// Mitsubishi GX Works2 project: project2 (1)   PLC: FX3G

// global labels: Global1
VAR_GLOBAL
  startday AT X007 : BOOL;
  lemonInput AT D1100 : REAL;
  raspberryInput AT D1110 : REAL;
  gummyBearInput AT D1130 : REAL;
  workLed AT Y007 : BOOL;
  fictivyStartday AT M5 : BOOL;
  emrgency AT X005 : BOOL;
  finishIngridiance AT M1 : BOOL;
  endDay AT M6 : BOOL;
  enoughIngredients AT M7 : BOOL;
  startDgima AT X001 : BOOL;
  analogInput1 AT D8280 : INT;
END_VAR
VAR_GLOBAL CONSTANT
  normalizationFactor : REAL := 400;
END_VAR
VAR_GLOBAL
  gumigumType AT D1502 : REAL;
  minRegularGumigum AT E0.0 : REAL;
  maxRegularGumigum AT E5.0 : REAL;
  regularGumigum AT M12 : BOOL;
  minPinukGumigum AT E6.0 : REAL;
  pinukGumigum AT M13 : BOOL;
  stabilizerInput AT D1120 : REAL;
END_VAR
VAR_GLOBAL CONSTANT
  minLemonRaspberryRegular : REAL := 35;
  minRaspberryRaspberryRegular : REAL := 280;
  minStabilizerRaspberryRegular : REAL := 35;
END_VAR
VAR_GLOBAL
  checkRaspberryRegular AT M2 : BOOL;
  checkLemonRegular AT M3 : BOOL;
END_VAR
VAR_GLOBAL CONSTANT
  minLemonLemonRegular : REAL := 420;
  minRaspberryLemonRegular : REAL;
  minStabilizerLemonRegular : REAL := 70;
  minLemonRaspberryPinuk : REAL := 105;
  minRaspberryRaspberryPinuk : REAL := 385;
  minStabilizerRaspberryPinuk : REAL := 70;
END_VAR
VAR_GLOBAL
  chechRaspberryPinuk AT M4 : BOOL;
END_VAR
VAR_GLOBAL CONSTANT
  minLemonLemonPinuk : REAL := 560;
  minRaspberryLemonPinuk : REAL;
  minStabilizerLemonPinuk : REAL := 140;
END_VAR
VAR_GLOBAL
  checkLemonPinuk AT M15 : BOOL;
  timer5Sec AT TC1 : BOOL;
END_VAR
VAR_GLOBAL CONSTANT
  fiveSec : INT := 50;
END_VAR
VAR_GLOBAL
  finishTimer AT TS1 : BOOL;
  iceCreamMaking AT Y000 : BOOL;
  coolContainer AT X002 : BOOL;
  timer8Sec AT TC3 : BOOL;
END_VAR
VAR_GLOBAL CONSTANT
  eightSec : INT := 80;
END_VAR
VAR_GLOBAL
  temp10Degrees AT X003 : BOOL;
  coolLed AT Y002 : BOOL;
END_VAR
VAR_GLOBAL CONSTANT
  gummyBearPinuk : REAL := 70;
  gummyBearRegular : REAL := 28;
END_VAR
VAR_GLOBAL
  onOffLed AT M16 : BOOL;
  timerRegularGummigum AT TC33 : BOOL;
END_VAR
VAR_GLOBAL CONSTANT
  OnOffRegular : INT := 30;
END_VAR
VAR_GLOBAL
  timerPinukGummigum AT TC55 : BOOL;
END_VAR
VAR_GLOBAL CONSTANT
  OnOffPinuk : INT := 50;
END_VAR
VAR_GLOBAL
  timerReset AT M17 : BOOL;
  timer1 AT TC10 : BOOL;
END_VAR
VAR_GLOBAL CONSTANT
  timeInterval : INT := 7;
END_VAR
VAR_GLOBAL
  endTimer1 AT TS10 : BOOL;
  mixingLedY5 AT Y005 : BOOL;
  mixingLedY6 AT Y006 : BOOL;
  timer2 AT TC20 : BOOL;
  endTimer2 AT TS20 : BOOL;
  packinIsOn AT X004 : BOOL;
  oneGummigumPack AT X000 : BOOL;
END_VAR
VAR_GLOBAL CONSTANT
  sevenCounter : INT := 7;
END_VAR
VAR_GLOBAL
  stillPacking AT TS8 : BOOL;
  finishToPack AT CS1 : BOOL;
  startCount AT CN1 : INT;
END_VAR
VAR_GLOBAL CONSTANT
  start1 : INT := 1;
  count6Pack : INT := 6;
END_VAR
VAR_GLOBAL
  finishPack AT Y004 : BOOL;
END_VAR
VAR_GLOBAL CONSTANT
  addPack : REAL := 1;
END_VAR
VAR_GLOBAL
  packCounter AT D1160 : REAL;
  printPack AT D1180 : REAL;
  analogOutput2 AT D8282 : INT;
  pinukForPack AT D1230 : REAL;
END_VAR
VAR_GLOBAL CONSTANT
  pinuk1260 : REAL := 1260;
  lemonPinuk665 : REAL := 665;
  raspberryPinuk385 : REAL := 385;
  stabilizerPinuk210 : REAL := 210;
  lemonRegular455 : REAL := 455;
  raspberryRegular280 : REAL := 280;
  stabilstabilizerRegular105 : REAL := 105;
END_VAR
VAR_GLOBAL
  regularForPack AT D1240 : REAL;
END_VAR
VAR_GLOBAL CONSTANT
  regular840 : REAL := 840;
END_VAR
VAR_GLOBAL
  coolRegularForPack AT D3040 : REAL;
  coolPinukForPack AT D3030 : REAL;
  endTimer8Sec AT TS3 : BOOL;
  mixpinukForPack AT D1330 : REAL;
  mixRegularForPack AT D1340 : REAL;
  timerPinukGummigum1 AT TS55 : BOOL;
  timerRegularGummigum1 AT TS33 : BOOL;
  resetCounter AT TC8 : BOOL;
END_VAR
VAR_GLOBAL CONSTANT
  resetCounter10 : INT := 10;
END_VAR
VAR_GLOBAL
  resetCounter1 AT TS8 : BOOL;
  pack7Gummigum AT CC1 : BOOL;
END_VAR
VAR_GLOBAL CONSTANT
  normalizationFactor400 : REAL := 40;
END_VAR

// task Task_01 (event TRUE, interval 0, priority 31): POU_01

PROGRAM POU_01
VAR CONSTANT
  checkRaspberryPinuk : BOOL;
END_VAR
(* structured ladder/FBD written out as ST: instructions are called as NAME(EN, inputs, outputs); _pN, _eN, _tN stand for wires *)
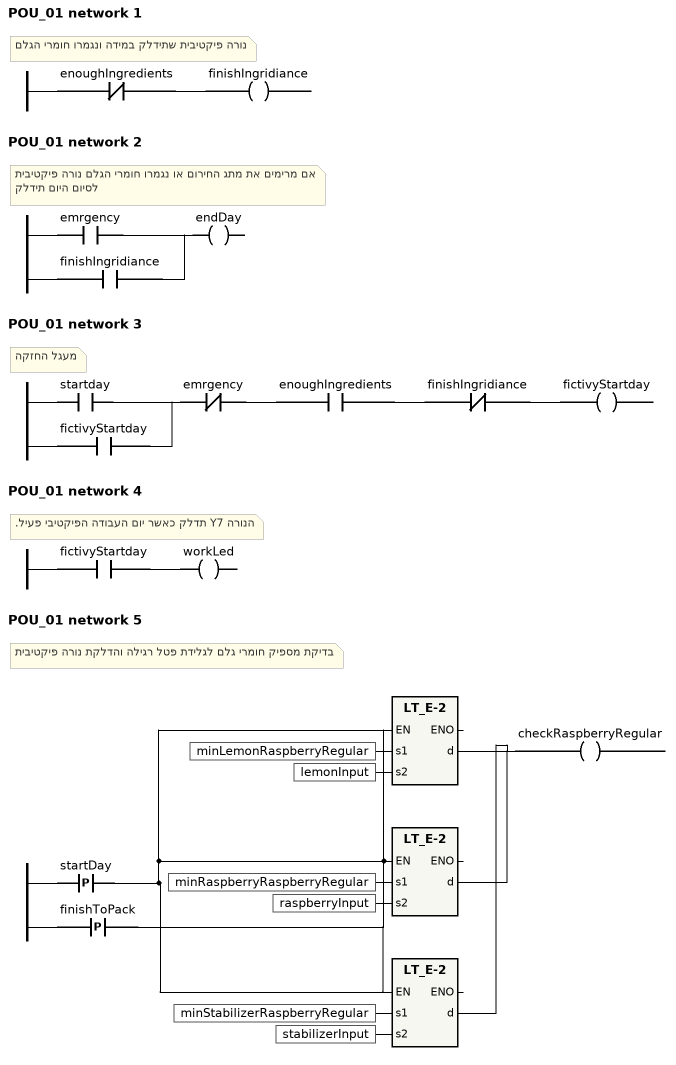
(* network 1 *)
(* נורה פיקטיבית שתידלק במידה ונגמרו חומרי הגלם *)
finishIngridiance := NOT enoughIngredients;
(* network 2 *)
(* אם מרימים את מתג החירום או נגמרו חומרי הגלם נורה פיקטיבית לסיום היום תידלק *)
endDay := emrgency OR finishIngridiance;
(* network 3 *)
(* מעגל החזקה *)
fictivyStartday := (((startday OR fictivyStartday) AND NOT emrgency) AND enoughIngredients) AND NOT finishIngridiance;
(* network 4 *)
(* הנורה Y7 תדלק כאשר יום העבודה הפיקטיבי פעיל. *)
workLed := fictivyStartday;
(* network 5 *)
(* בדיקת מספיק חומרי גלם לגלידת פטל רגילה והדלקת נורה פיקטיבית *)
_p1 := LDP(TRUE, startDay) OR LDP(TRUE, finishToPack);
LT_E(_p1, minLemonRaspberryRegular, lemonInput, _t2);
LT_E(_p1, minRaspberryRaspberryRegular, raspberryInput, _t3);
LT_E(_p1, minStabilizerRaspberryRegular, stabilizerInput, _t4);
checkRaspberryRegular := _t2 OR _t3 OR _t4;
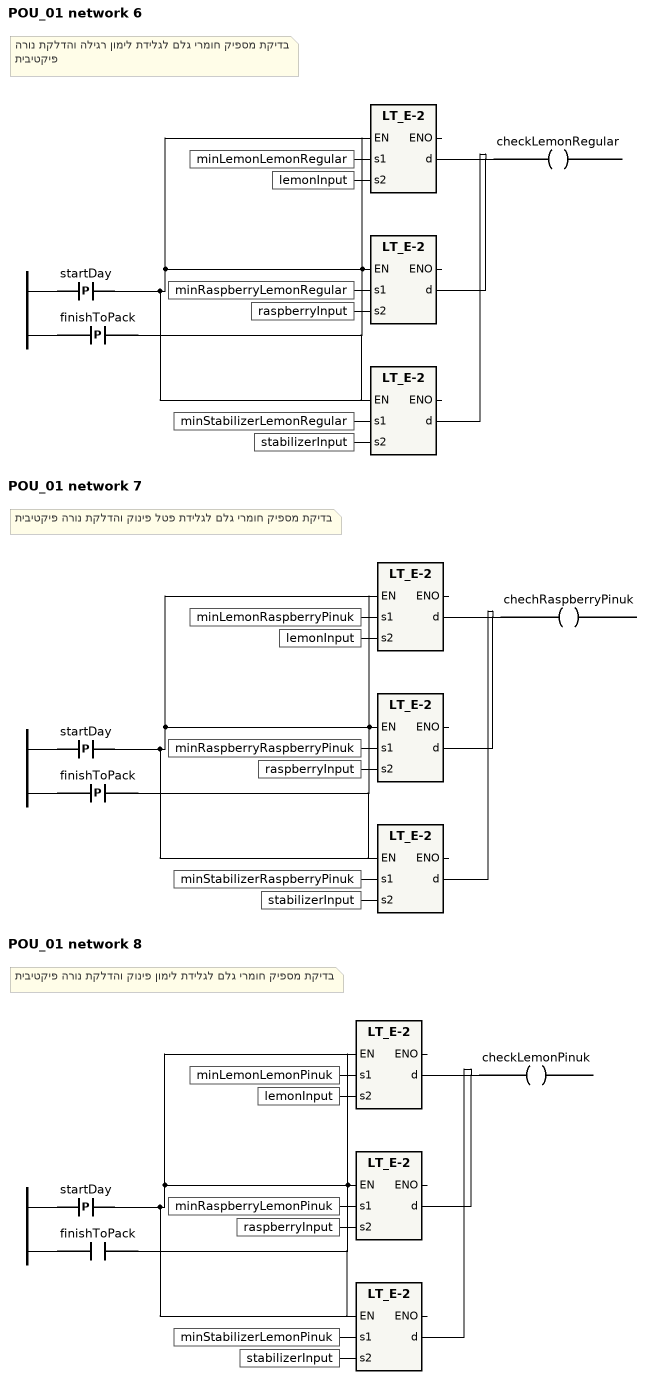
(* network 6 *)
(* בדיקת מספיק חומרי גלם לגלידת לימון רגילה והדלקת נורה פיקטיבית *)
_p1 := LDP(TRUE, startDay) OR LDP(TRUE, finishToPack);
LT_E(_p1, minLemonLemonRegular, lemonInput, _t2);
LT_E(_p1, minRaspberryLemonRegular, raspberryInput, _t3);
LT_E(_p1, minStabilizerLemonRegular, stabilizerInput, _t4);
checkLemonRegular := _t2 OR _t3 OR _t4;
(* network 7 *)
(* בדיקת מספיק חומרי גלם לגלידת פטל פינוק והדלקת נורה פיקטיבית *)
_p1 := LDP(TRUE, startDay) OR LDP(TRUE, finishToPack);
LT_E(_p1, minLemonRaspberryPinuk, lemonInput, _t2);
LT_E(_p1, minRaspberryRaspberryPinuk, raspberryInput, _t3);
LT_E(_p1, minStabilizerRaspberryPinuk, stabilizerInput, _t4);
chechRaspberryPinuk := _t2 OR _t3 OR _t4;
(* network 8 *)
(* בדיקת מספיק חומרי גלם לגלידת לימון פינוק והדלקת נורה פיקטיבית *)
_p1 := LDP(TRUE, startDay) OR finishToPack;
LT_E(_p1, minLemonLemonPinuk, lemonInput, _t2);
LT_E(_p1, minRaspberryLemonPinuk, raspberryInput, _t3);
LT_E(_p1, minStabilizerLemonPinuk, stabilizerInput, _t4);
checkLemonPinuk := _t2 OR _t3 OR _t4;
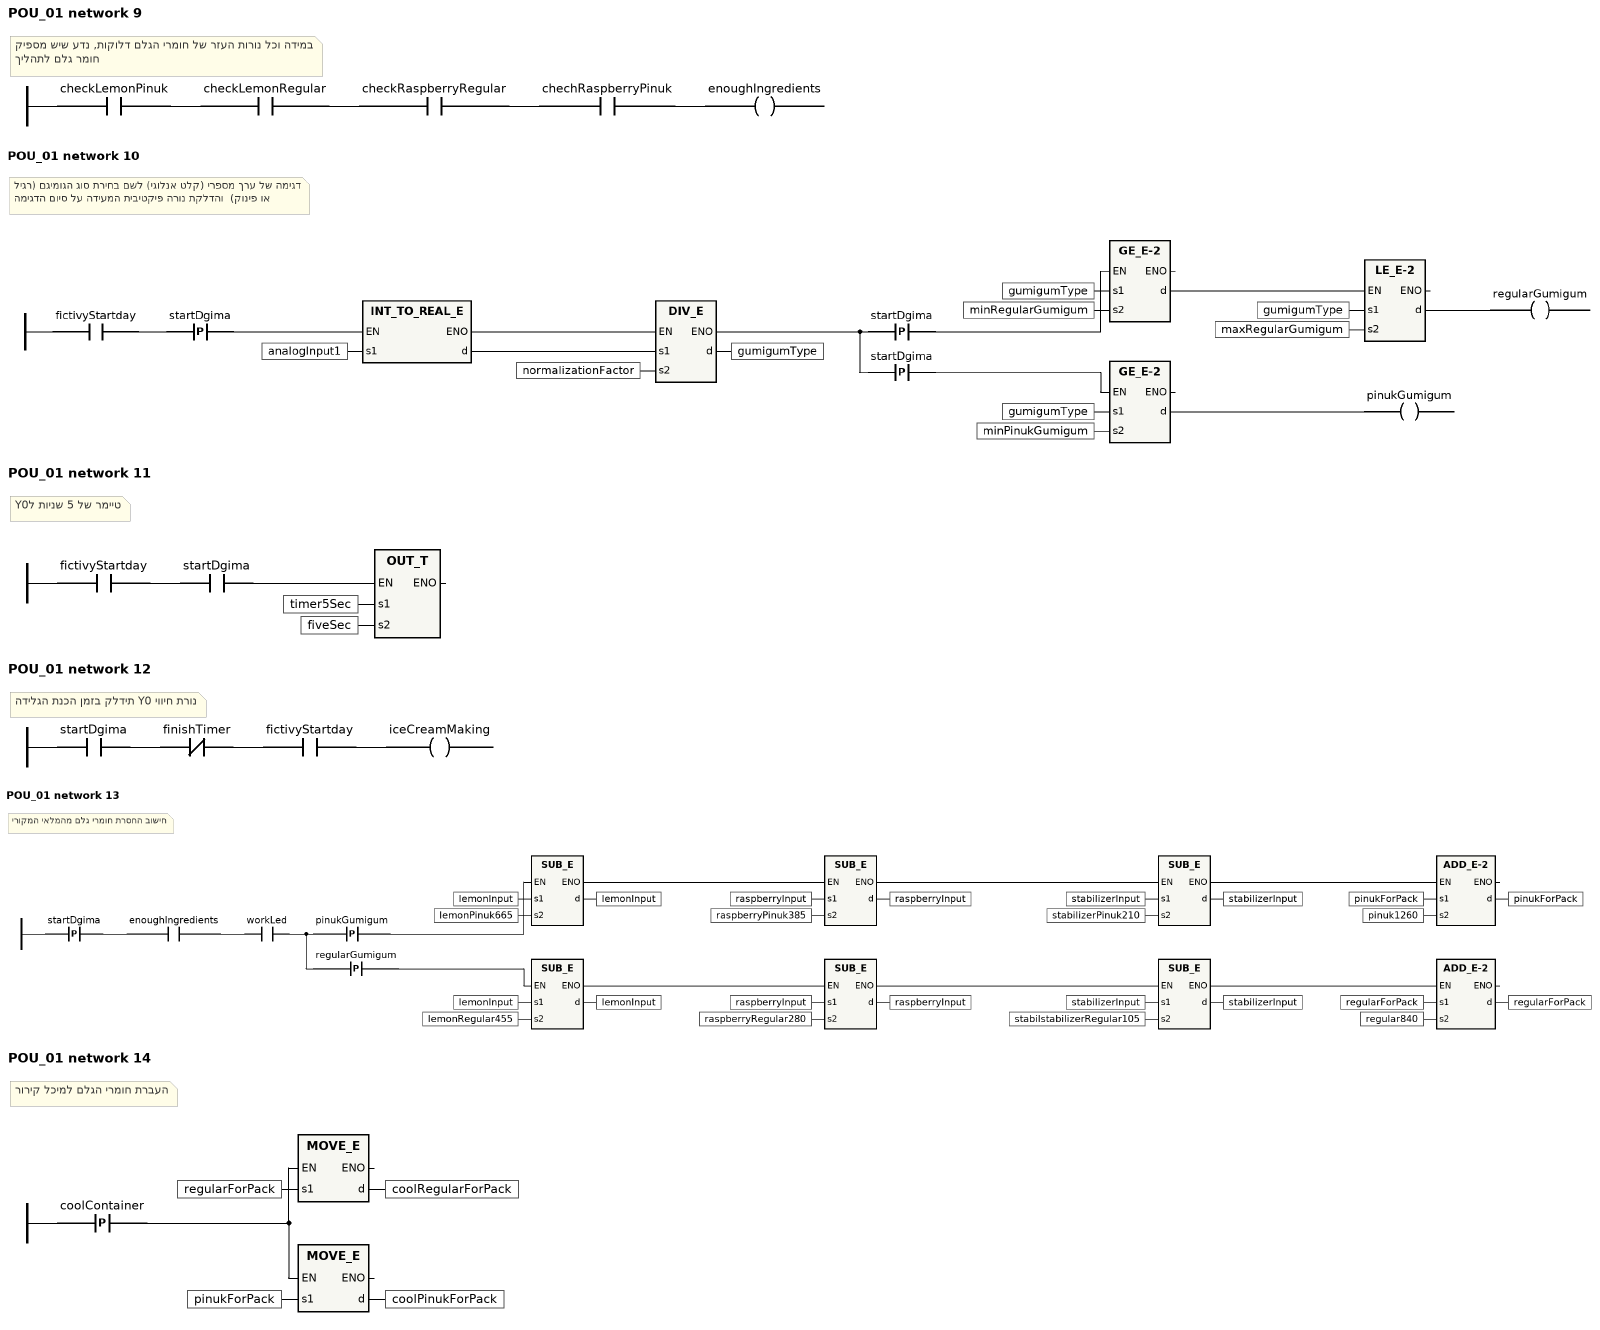
(* network 9 *)
(* במידה וכל נורות העזר של חומרי הגלם דלוקות, נדע שיש מספיק חומר גלם לתהליך *)
enoughIngredients := checkLemonPinuk AND checkLemonRegular AND checkRaspberryRegular AND chechRaspberryPinuk;
(* network 10 *)
(* דגימה של ערך מספרי (קלט אנלוגי) לשם בחירת סוג הגומיגם (רגיל או פינוק)  והדלקת נורה פיקטיבית המעידה על סיום הדגימה *)
_e2 := INT_TO_REAL_E(fictivyStartday AND LDP(TRUE, startDgima), analogInput1, _t1);
_e3 := DIV_E(_e2, _t1, normalizationFactor, gumigumType);
GE_E(_e3 AND LDP(TRUE, startDgima), gumigumType, minRegularGumigum, _t4);
LE_E(_t4, gumigumType, maxRegularGumigum, _t5);
regularGumigum := _t5;
GE_E(_e3 AND LDP(TRUE, startDgima), gumigumType, minPinukGumigum, _t6);
pinukGumigum := _t6;
(* network 11 *)
(* טיימר של 5 שניות לY0 *)
OUT_T(fictivyStartday AND startDgima, timer5Sec, fiveSec);
(* network 12 *)
(* נורת חיווי Y0 תידלק בזמן הכנת הגלידה *)
iceCreamMaking := startDgima AND NOT finishTimer AND fictivyStartday;
(* network 13 *)
(* חישוב החסרת חומרי גלם מהמלאי המקורי *)
_p1 := LDP(TRUE, startDgima) AND enoughIngredients AND workLed;
_e2 := SUB_E(_p1 AND LDP(TRUE, pinukGumigum), lemonInput, lemonPinuk665, lemonInput);
_e3 := SUB_E(_e2, raspberryInput, raspberryPinuk385, raspberryInput);
_e4 := SUB_E(_e3, stabilizerInput, stabilizerPinuk210, stabilizerInput);
ADD_E(_e4, pinukForPack, pinuk1260, pinukForPack);
_e5 := SUB_E(_p1 AND LDP(TRUE, regularGumigum), lemonInput, lemonRegular455, lemonInput);
_e6 := SUB_E(_e5, raspberryInput, raspberryRegular280, raspberryInput);
_e7 := SUB_E(_e6, stabilizerInput, stabilstabilizerRegular105, stabilizerInput);
ADD_E(_e7, regularForPack, regular840, regularForPack);
(* network 14 *)
(* העברת חומרי הגלם למיכל קירור *)
_p1 := LDP(TRUE, coolContainer);
MOVE_E(_p1, regularForPack, coolRegularForPack);
MOVE_E(_p1, pinukForPack, coolPinukForPack);
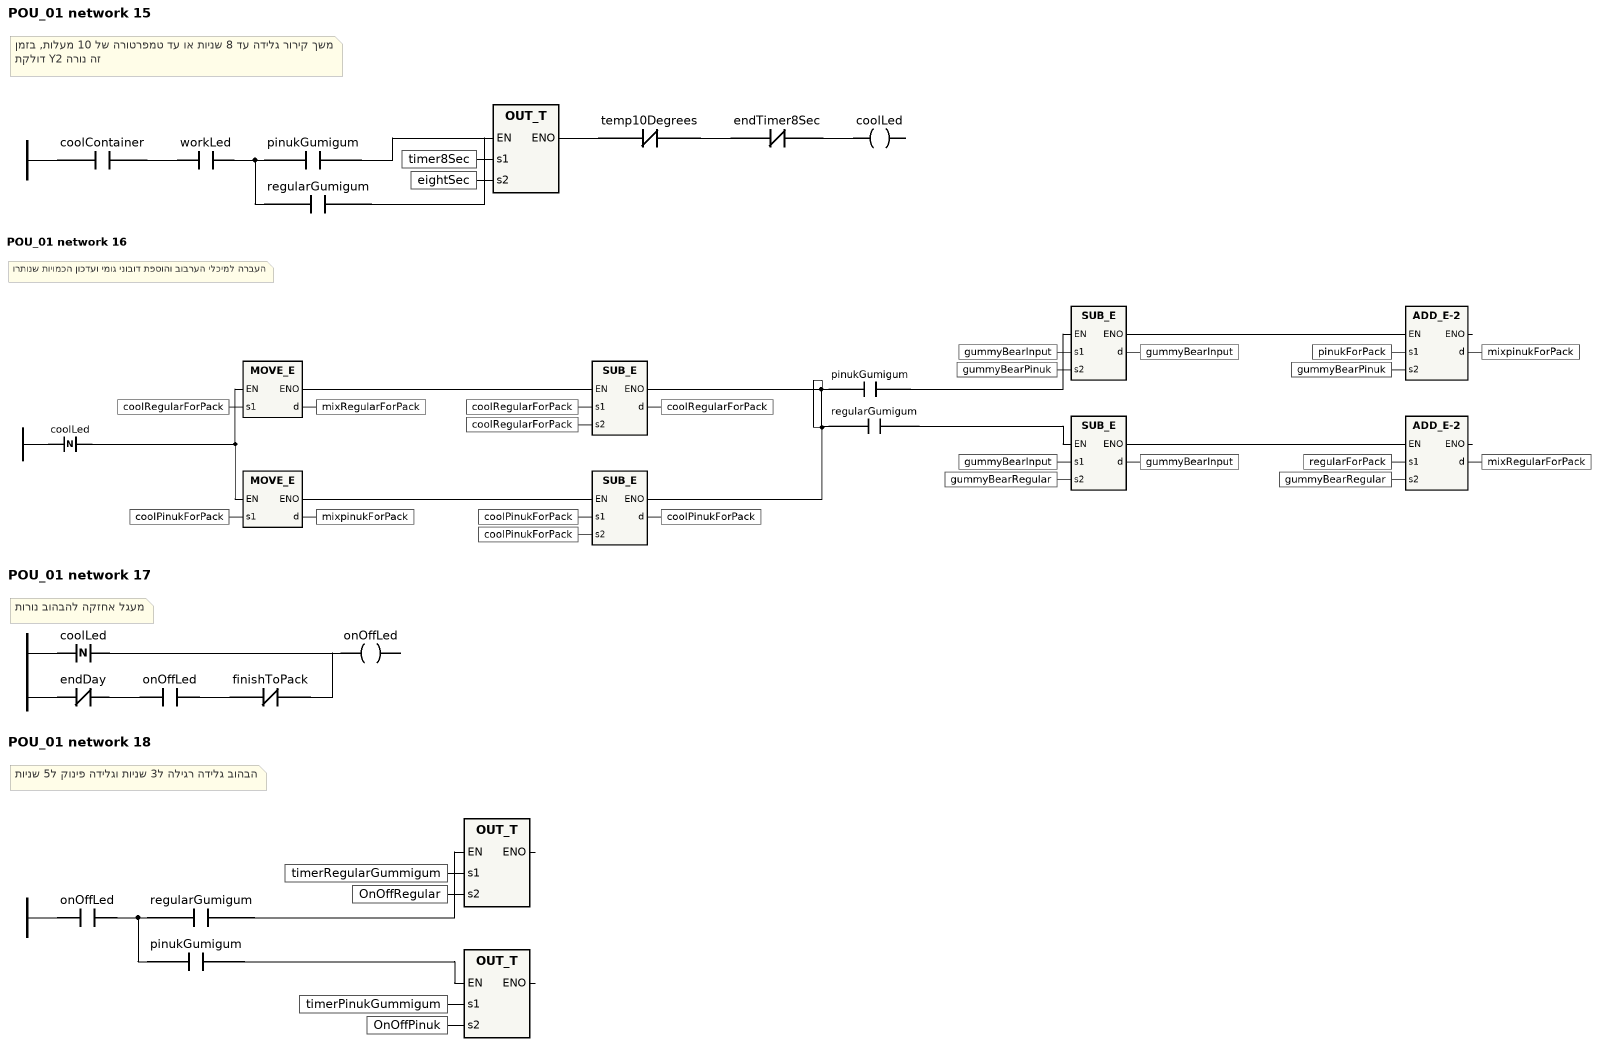
(* network 15 *)
(* משך קירור גלידה עד 8 שניות או עד טמפרטורה של 10 מעלות, בזמן זה נורה Y2 דולקת *)
_p1 := coolContainer AND workLed;
_e2 := OUT_T((_p1 AND pinukGumigum) OR (_p1 AND regularGumigum), timer8Sec, eightSec);
coolLed := _e2 AND NOT temp10Degrees AND NOT endTimer8Sec;
(* network 16 *)
(* העברה למיכלי הערבוב והוספת דובוני גומי ועדכון הכמויות שנותרו *)
_p1 := LDF(TRUE, coolLed);
_e2 := MOVE_E(_p1, coolRegularForPack, mixRegularForPack);
_e3 := SUB_E(_e2, coolRegularForPack, coolRegularForPack, coolRegularForPack);
_e4 := MOVE_E(_p1, coolPinukForPack, mixpinukForPack);
_e5 := SUB_E(_e4, coolPinukForPack, coolPinukForPack, coolPinukForPack);
_p6 := _e3 OR _e5;
_e7 := SUB_E(_p6 AND pinukGumigum, gummyBearInput, gummyBearPinuk, gummyBearInput);
ADD_E(_e7, pinukForPack, gummyBearPinuk, mixpinukForPack);
_e8 := SUB_E(_p6 AND regularGumigum, gummyBearInput, gummyBearRegular, gummyBearInput);
ADD_E(_e8, regularForPack, gummyBearRegular, mixRegularForPack);
(* network 17 *)
(* מעגל אחזקה להבהוב נורות *)
onOffLed := LDF(TRUE, coolLed) OR (NOT endDay AND onOffLed AND NOT finishToPack);
(* network 18 *)
(* הבהוב גלידה רגילה ל3 שניות וגלידה פינוק ל5 שניות *)
OUT_T(onOffLed AND regularGumigum, timerRegularGummigum, OnOffRegular);
OUT_T(onOffLed AND pinukGumigum, timerPinukGummigum, OnOffPinuk);
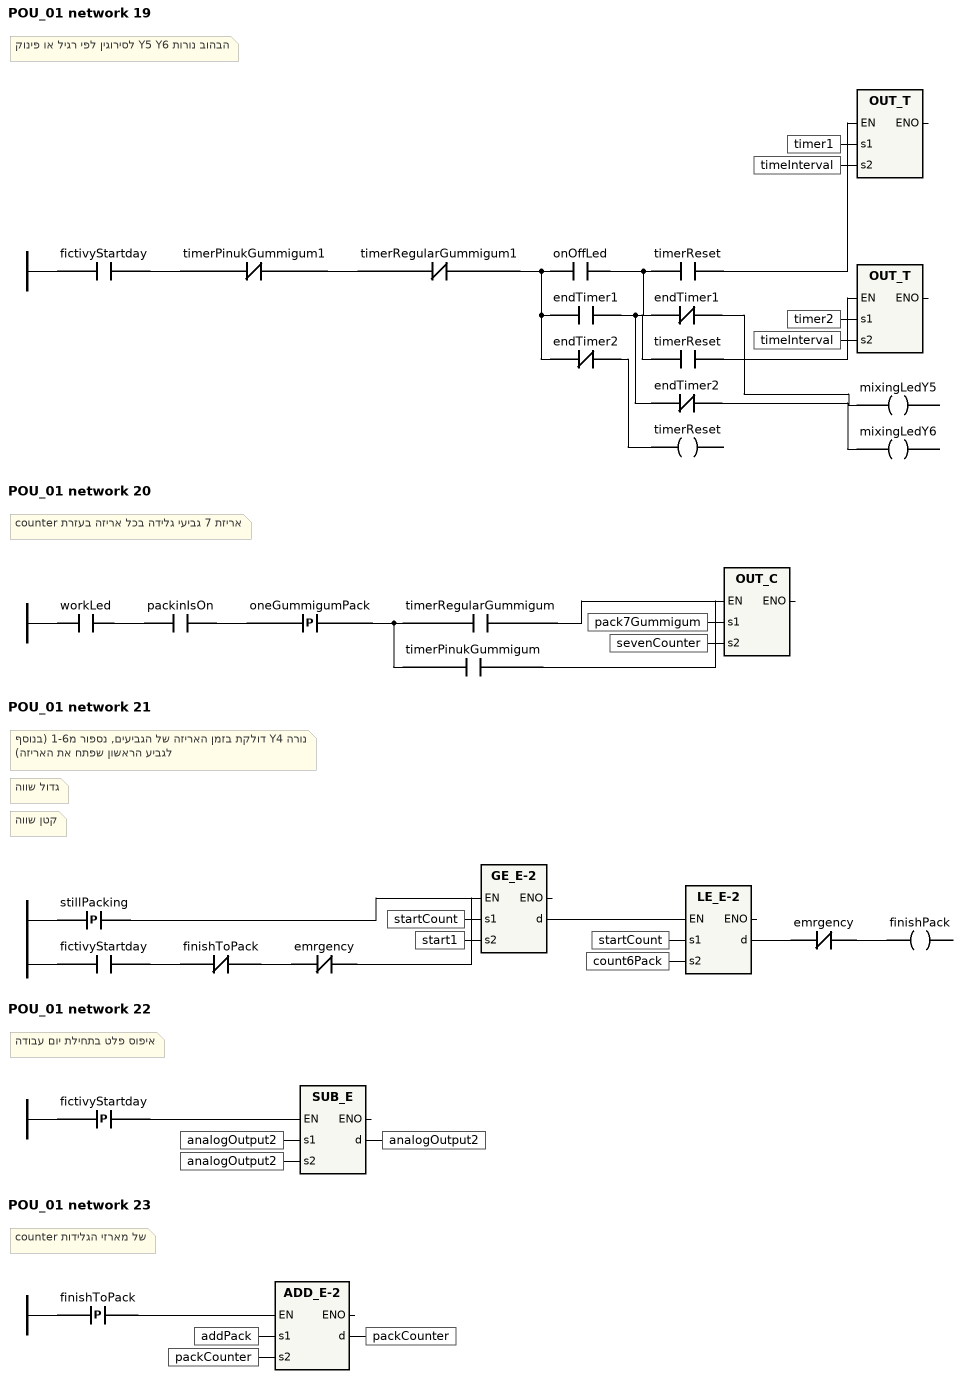
(* network 19 *)
(* הבהוב נורות Y5 Y6 לסירוגין לפי רגיל או פינוק *)
_p1 := fictivyStartday AND NOT timerPinukGummigum1 AND NOT timerRegularGummigum1;
_p2 := _p1 AND onOffLed;
OUT_T(_p2 AND timerReset, timer1, timeInterval);
mixingLedY5 := _p2 AND NOT endTimer1;
_p3 := _p1 AND endTimer1;
OUT_T(_p3 AND timerReset, timer2, timeInterval);
mixingLedY6 := _p3 AND NOT endTimer2;
timerReset := _p1 AND NOT endTimer2;
(* network 20 *)
(* אריזת 7 גביעי גלידה בכל אריזה בעזרת counter *)
_p1 := workLed AND packinIsOn AND LDP(TRUE, oneGummigumPack);
OUT_C((_p1 AND timerRegularGummigum) OR (_p1 AND timerPinukGummigum), pack7Gummigum, sevenCounter);
(* network 21 *)
(* נורה Y4 דולקת בזמן האריזה של הגביעים, נספור מ1-6 (בנוסף לגביע הראשון שפתח את האריזה) *)
(* גדול שווה *)
(* קטן שווה *)
GE_E(LDP(TRUE, stillPacking) OR (fictivyStartday AND NOT finishToPack AND NOT emrgency), startCount, start1, _t1);
LE_E(_t1, startCount, count6Pack, _t2);
finishPack := _t2 AND NOT emrgency;
(* network 22 *)
(* איפוס פלט בתחילת יום עבודה *)
SUB_E(LDP(TRUE, fictivyStartday), analogOutput2, analogOutput2, analogOutput2);
(* network 23 *)
(* counter של מארזי הגלידות *)
ADD_E(LDP(TRUE, finishToPack), addPack, packCounter, packCounter);
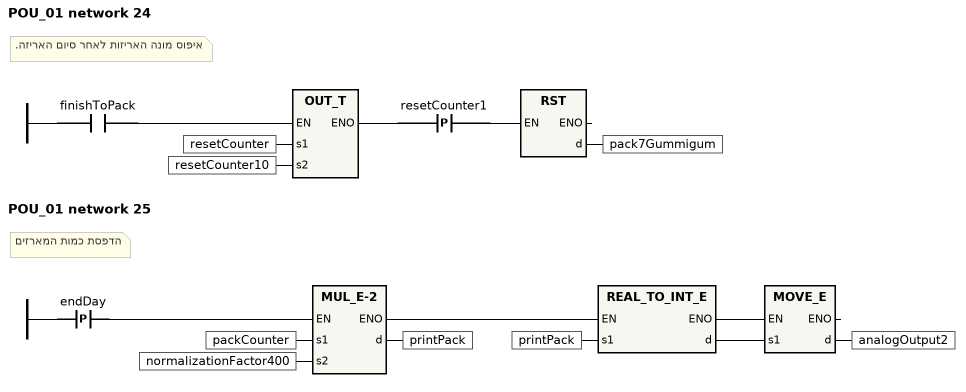
(* network 24 *)
(* איפוס מונה האריזות לאחר סיום האריזה. *)
_e1 := OUT_T(finishToPack, resetCounter, resetCounter10);
RST(_e1 AND LDP(TRUE, resetCounter1), pack7Gummigum);
(* network 25 *)
(* הדפסת כמות המארזים *)
_e1 := MUL_E(LDP(TRUE, endDay), packCounter, normalizationFactor400, printPack);
_e3 := REAL_TO_INT_E(_e1, printPack, _t2);
MOVE_E(_e3, _t2, analogOutput2);
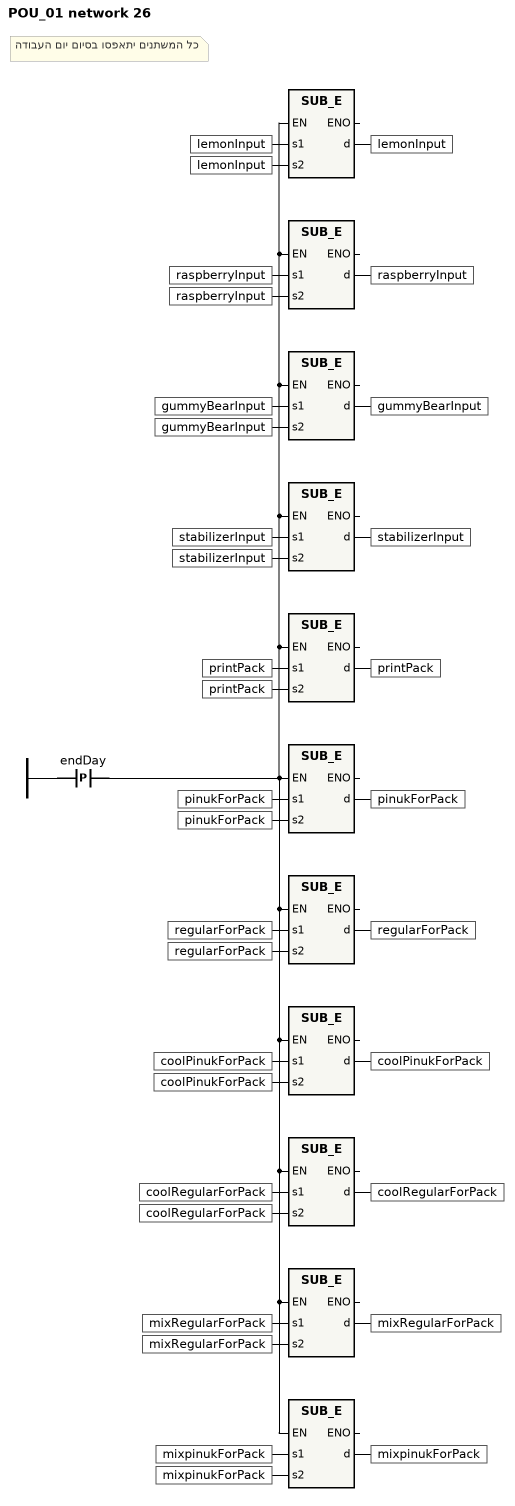
(* network 26 *)
(* כל המשתנים יתאפסו בסיום יום העבודה *)
_p1 := LDP(TRUE, endDay);
SUB_E(_p1, lemonInput, lemonInput, lemonInput);
SUB_E(_p1, raspberryInput, raspberryInput, raspberryInput);
SUB_E(_p1, gummyBearInput, gummyBearInput, gummyBearInput);
SUB_E(_p1, stabilizerInput, stabilizerInput, stabilizerInput);
SUB_E(_p1, printPack, printPack, printPack);
SUB_E(_p1, pinukForPack, pinukForPack, pinukForPack);
SUB_E(_p1, regularForPack, regularForPack, regularForPack);
SUB_E(_p1, coolPinukForPack, coolPinukForPack, coolPinukForPack);
SUB_E(_p1, coolRegularForPack, coolRegularForPack, coolRegularForPack);
SUB_E(_p1, mixRegularForPack, mixRegularForPack, mixRegularForPack);
SUB_E(_p1, mixpinukForPack, mixpinukForPack, mixpinukForPack);
END_PROGRAM
